Universal Robots PolyScope program: g01_cycle.urp

Program g01_cycle (installation=default directory=/programs createdIn=5.9.1.1031110 lastSavedIn=5.9.1.1031110 robotSerialNumber=20195501059)
Calibrated DH parameters: a=[0.000146, -0.418764, -0.053981, 0.000058, -0.000023, 0]; d=[0.162545, 37.319448, -206.067439, 168.881546, 0.09955, 0.099464]; alpha=[1.57004, -0.001979, 0.002304, 1.570607, -1.57066, 0]; deltaTheta=[0, -0.174616, -1.258233, 1.432844, -0.000001, 0]
Robot Program (runOnlyOnce=true)
  URCap Grip Check (Robotiq_Grippers, Robotiq Inc.) dataModel(ObjectDetectedKey=true, DimensionValidationKey=false, DimensionKey=100.0, DimensionDimensionPositiveGapKey=5.0, DimensionNegativeGapKey=5.0, GripperIdKey=1, ModelDefinedKey=true); state(isChildrenLocked=true)
    URCap If (Robotiq_Grippers, Robotiq Inc.)
      Call g01_nut_dropoff
  Call g01_home_s
  Call g01_nut_pickup_1
  Call g01_apply
  URCap Grip Check (Robotiq_Grippers, Robotiq Inc.) dataModel(ObjectDetectedKey=true, DimensionValidationKey=false, DimensionKey=100.0, DimensionDimensionPositiveGapKey=5.0, DimensionNegativeGapKey=5.0, GripperIdKey=1, ModelDefinedKey=true); state(isChildrenLocked=true)
    URCap If (Robotiq_Grippers, Robotiq Inc.)
      Call g01_nut_dropoff
  Call g01_home_s
SubProgram  [hidden by the author, left out]
SubProgram  [hidden by the author, left out]
SubProgram  [hidden by the author, left out]
SubProgram  [hidden by the author, left out]
SubProgram g01_nut_dropoff [hidden by the author, left out]
SubProgram g01_home_s [hidden by the author, left out]
SubProgram g01_nut_pickup_1 [hidden by the author, left out]
SubProgram g01_apply [hidden by the author, left out]
